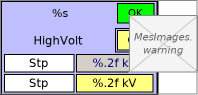
VISUALIZATION VISU_HT_CANON_ST10  // 198x95
VAR_IN_OUT
	m_Input_SOURCE : BLOCK_CANON_ST10;
END_VAR
    Rectangle (0,0 158x95)
    Rectangle (3,30 110x21), "HighVolt"
    Rectangle (117,3 37x20), "NOK", invisible if: NOT m_Input_SOURCE.STATE_NOK
    Rectangle (117,30 37x20), "OFF", invisible if: m_Input_SOURCE.STATE_HV OR m_Input_SOURCE.STATE_HV_ON
    Rectangle (117,3 37x20), "OK", invisible if: m_Input_SOURCE.STATE_NOK
    Rectangle (117,30 37x20), "ON", invisible if: NOT m_Input_SOURCE.STATE_HV AND NOT m_Input_SOURCE.STATE_HV_ON
    RoundedRectangle (4,54 70x18), "Stp", invisible if: Global_Variables.MACHINE.State_manu
    RoundedRectangle (76,54 77x18), "%.2f kV", text variable: m_Input_SOURCE.AO_QUHV.Value, invisible if: Global_Variables.MACHINE.State_manu
    Rectangle (117,30 37x20), "ON", invisible if: m_Input_SOURCE.STATE_HV_ON OR NOT m_Input_SOURCE.STATE_HV
    Rectangle (0,3 120x21), "%s", text variable: m_Input_SOURCE.MNEMO
    Polyline (7,35)
    RoundedRectangle (4,74 70x18), "Stp", invisible if: NOT Global_Variables.PRG_USER.ACTU_USER.MAINTENANCE OR NOT MACHINE.State_manu
    RoundedRectangle (76,74 77x18), "%.2f kV", text variable: m_Input_SOURCE.PRM_TENSION, invisible if: NOT Global_Variables.PRG_USER.ACTU_USER.MAINTENANCE OR NOT MACHINE.STATE_Manu
        OnMouseDown: write the text variable via InputWithLimits, min 7, max 10
    Rectangle (115,28 41x24), invisible if: NOT m_Input_SOURCE.HV.AUTOR_ON_IHM AND NOT m_Input_SOURCE.HV.AUTOR_OFF_IHM, input disabled if: (NOT m_Input_SOURCE.HV.AUTOR_ON_IHM AND NOT m_Input_SOURCE.HV.AUTOR_OFF_IHM) OR NOT PRG_User.ACTU_USER.MAINTENANCE
        tap m_Input_SOURCE.HV.M_On
    Image (129,15 69x57), invisible if: NOT m_Input_SOURCE.STATE_NOK, image: MesImages.warning
END_VISUALIZATION

(* stored: Version 1.1.0.1, ProductVersion 3.1.4024.10
   Visu VISU_HT_CANON_ST10: Id {ae73b106-1340-41af-a58c-f59707eddd1e} *)
